TYPE ST_IO2_OutputPLC :
STRUCT
	bOutputEnable				: BOOL;

	bStateOutput				: BOOL;
	bDelayedOutput			: BOOL;
	bLockedOutput			: BOOL;
	bDelayedLockedOtput		: BOOL;
END_STRUCT
END_TYPE

(* stored: Version 1.1.0.1, ProductVersion 3.1.4024.15
   DUT ST_IO2_OutputPLC: Id {19ac6cb9-5832-4fd4-a4d0-6e2639ea754f} *)
